// TIA Portal V16 export
// export: Created 2021-08-30T11:09:35.4904Z, ExportSetting WithDefaults, DisplayName Totally Integrated Automation Portal, DisplayVersion V16 Update 3, DisplayName TIA Portal Version Control Interface, DisplayVersion V16 Update 2, DisplayName TIA Portal Openness, DisplayVersion V16 Update 3, DisplayName TIA Portal Teamcenter Gateway, DisplayVersion V16, DisplayName STEP 7 Professional, DisplayVersion V16 Update 3, DisplayName STEP 7 Safety, DisplayVersion V16, DisplayName WinCC Advanced, DisplayVersion V16 Update 3
DATA_BLOCK "AllPump_DB"   // DB9
VERSION : 0.1
// stored: AutoNumber true, DBAccessibleFromOPCUA true, InstanceOfName AllPump, InstanceOfType FB
"AllPump"
   // VAR
   //    PU30x { S7_SetPoint := 'True'} : "PumpCntrl2Pu1Fc";
   //    cmUZ1 { S7_SetPoint := 'True'} : Bool;
   //    tmrLowPresP30x { S7_SetPoint := 'True'} : TON_TIME;
   //    tmrLowFreqP30x { S7_SetPoint := 'True'} : TON_TIME;
   //    tLowPresP30x { S7_SetPoint := 'True'} : Time;
   //    tLowFreqP30x : Time;
   // END_VAR
BEGIN
END_DATA_BLOCK
